{attribute 'qualified_only'}
VAR_GLOBAL
	// Schnittstellenvariablen 
		// System: 
		SystemState								:eSystemState; 
		SystemCommand							:eSystemCommand; 
		ErrorID									:INT;
		
		// Kontrollvariablen: 
		Reset									:BOOL;
		Execute									:BOOL;
		
		// Prozessvariablen
		eKraftLimitValue						:sKraftVariablen;
		eKraftErreichtValue						:sKraftVariablen;
		
		
		// SkillStates
		
		// ObjectStates
		Robot_State								:eObjectAktorState;
		Greifer_State							:eObjectAktorState;
		Sensor_State							:eObjectSensorState;
END_VAR

(* stored: Version 1.1.0.1
   GVL GVL: Id {c71acb86-7d2e-4817-95ad-fa2de8d14b8a} *)
